PROGRAM POU
VAR
END_VAR

END_PROGRAM

(* stored: Version 1.1.0.1, ProductVersion 3.1.4022.18
   POU POU: Id {f0ddbdc8-838d-44b9-8b6f-54afc3e17411}, SpecialFunc None *)
